FUNCTION_BLOCK AnalogOutput IMPLEMENTS I_AnalogOutput
VAR_INPUT
END_VAR
VAR_OUTPUT
END_VAR
VAR
	ID:				STRING(25);
	Output			AT%I*: INT;
	fOffset:		LREAL;
	fMaximum:		LREAL;
END_VAR

METHOD FB_init : BOOL
VAR_INPUT
	bInitRetains : BOOL; // if TRUE, the retain variables are initialized (warm start / cold start)
	bInCopyCode : BOOL;  // if TRUE, the instance afterwards gets moved into the copy code (online change)
	ID:				STRING(25);
	fOffset:		LREAL;
	fMaximum:		LREAL;
END_VAR
THIS^.ID:= ID;
THIS^.fOffset:= fOffset;
THIS^.fMaximum:= fMaximum;
END_METHOD

PROPERTY PUBLIC P_ID : String(25)
GET
P_ID:= ID;
END_GET
END_PROPERTY

PROPERTY PUBLIC P_Value : Lreal
SET // PUBLIC
Output:= LREAL_TO_INT(P_Value);
END_SET
END_PROPERTY

END_FUNCTION_BLOCK

(* stored: Version 1.1.0.1
   POU AnalogOutput: Id {7f986a17-ab6d-03bd-1c98-a964e10e1b1e}, SpecialFunc None
   Method FB_init: Id {fc427ba8-2be8-0fc8-1ba1-4c059d06ed11}
   Property P_ID: Id {030e0eaa-c0a4-09b4-3514-eb98d5fd7097}
   Get Get: Id {25c131a6-5f18-024c-3a39-ec1eed18a7fb}
   Property P_Value: Id {a955e2d0-0b5a-083c-1316-087f566ed02a}
   Set Set: Id {55ec4fbd-3d98-0de0-2d45-228ab7d2678e} *)
